{attribute 'linkalways'}
INTERFACE Startable EXTENDS __SYSTEM.IQueryInterface

METHOD Start : CommandStatus
END_METHOD

END_INTERFACE

(* stored: Version 1.1.0.1, ProductVersion 3.1.4024.15
   Itf Startable: Id {340a0c3d-feb4-48a0-ac72-cfe9dee7ee75}
   Method Start: Id {7e4dc126-77fa-4b6a-ba6c-f59aa52f4abb} *)
